Staubli VAL3: pasteItem.pgx

public program pasteItem(num& x_nIndex[] (dimensions=1))
  local num l_nSize
  local num i
  local InstrItem l_sItem
  local num l_nTemp
  local string l_sRight
begin
  call getSizeItem(l_nSize)
  l_nTemp=x_nIndex+1
  for i=0 to (l_nSize-1)
    call getItem(l_sItem,i)
    if find(l_sItem.sType,"#")!=-1
      if l_nTemp<=i
        i=i+1
      endIf
      l_sItem.sType=right(l_sItem.sType,len(l_sItem.sType)-1)
      call insertItem(l_sItem,l_nTemp)
      l_nTemp=l_nTemp+1
      l_nSize=l_nSize+1
    endIf
  endFor
  // unselect all
  call unSelectItem()
end
